FUNCTION_BLOCK FB_ModuleLogger IMPLEMENTS I_Logger
VAR
END_VAR

METHOD M_Log
VAR_INPUT
	stEvent	: 		ST_Event;
END_VAR
END_METHOD

END_FUNCTION_BLOCK

(* stored: Version 1.1.0.1, ProductVersion 3.1.4024.12
   POU FB_ModuleLogger: Id {a6fc589b-3f77-0dc8-1c02-65bea2758222}, SpecialFunc None
   Method M_Log: Id {ff8b0304-c1ca-062b-059f-da74ab423126} *)
